(*
Nazwa:			FB_WickFeederStation
Opis:			Podajnik knotów
Wersja:			v1.0
Data:			2025-12-29
Autor:			MK
Urzadzenia:		Podnosnik stacji, grzałka, czujnik temp, ssawka
Konfiguracja:	
Info: 
*)




FUNCTION_BLOCK FB_WickFeederStation
VAR_INPUT
	_CONTROL_:BOOL;	
	bEnable:BOOL;					//Zezowlenie na pracę podajnika knotów
	bEStop:BOOL;					//Stop awaryjny nieaktywny
	bRun:BOOL;						//Zezwolenie na podanie knotów do wbijaków - jak maszyna w Execute musi być na 1
	bRun1: BOOL;					//Zezwolenie na wbicie knota
	bRun2: BOOL;					//Zezwolenie na wbicie knota
	bHoming:BOOL;					//Zezwolenie na wykonanie bazowania i pozycjonowania podajnika
	bHeightSet:BOOL;				//Ustaw wysokość
	bIgnoreError:BOOL;				//Ignorowania błędów cyklu pracy
	bReset:BOOL;					//Reset błędu, jeśli w stanie "eError"
	lrPositionHeightSV:LREAL;		//Wysokość zadana na której ma znajdować się podajnik
	lrMaxHeight:LREAL;				//Maksymalna wysokość podajnika platynek
	lrMinHeight:LREAL;				//Minimalna wysokość podajnika platynek
	bManualMovement:BOOL; 			//Uruchomienie trybu ruchów ręcznych
	
	_SENSORS_:BOOL;	
	bWheelLevelSensor			: BOOL;	
	bWheelSensor				: BOOL;
	bQueFullAfterWheelSensor	: BOOL;			//Czujnik zapełnienia rękawa
	bQueFullSensor				: BOOL;			//Czujnik zapełnienia rękawa
	bWickAtPipe					: BOOL;			//Czujnik na końcu rękawa
	bSeparatorPos1				: BOOL;			//Separator nad torem 1
	bSeparatorPos2				: BOOL;			//Separator nad torem 2
	bQueFullAtSleve1			: BOOL;			//Czujnik zapełnienia rękawa 1
	bQueFullAtSleve2			: BOOL;			//Czujnik zapełnienia rękawa 2
	bWickAtSleve1				: BOOL;			//Czujnik na końcu rękawa 1
	bWickAtSleve2				: BOOL;			//Czujnik na końcu rękawa 2
	bSleve1SeparatorIn			: BOOL;			//Separator pod rękawem
	bSleve1SeparatorOut			: BOOL;			//Separator nad butelką
	bSleve2SeparatorIn			: BOOL;			//Separator pod rękawem
	bSleve2SeparatorOut			: BOOL;			//Separator nad butelką
	bHammer1Up					: BOOL;			//Wbijak pozycja górna
	bHammer1Down				: BOOL;			//Wbijak pozycja dolna
	bHammer2Up					: BOOL;			//Wbijak pozycja górna
	bHammer2Down				: BOOL;			//Wbijak pozycja dolna
	bFormPositioningHide1		: BOOL;			//Wbijak pozycja dolna
	bFormPositioningHide2		: BOOL;			//Wbijak pozycja dolna
	
	_HEIGHTMOTOR_ :BOOL;	
	udiHeightMotorEncoderCV		: UDINT;		//Sygnał impulsów enkodera siłownika
	bHeightEncoderSetCDone		: BOOL;	
	rHeightMotorPositionOffset 	: REAL;			//Wysokość bazowani podnośnika
//	nPositionHeightCV			: LREAL;		//Aktualna wysokość podajnika platynek
	
	_BOWLMOTOR_ :BOOL;
	bEngineOK					: BOOL;					//Wejście czujnika zabezpieczenia silnika 
	InEngineVelocityCV 			: UDINT;		
	InEngineSTW 				: UINT; 				// Statusword transportera wejściowo wyjściowego
	IbEngineWcState				: BOOL; 				// Statusword transportera wejściowo wyjściowego
	_PARAMETERS_:BOOL;
	iTimeDelayOn				: INT; 					//Czas na właczenie silnika sortera po zaniku sygnału przepełnienia z rękawa
	iTimeDelayOff				: INT; 					// Czas na wylączenie silnika sortera po wykryciu sygnału przepełnienia z rękawa sortera
	iTimeToEmptySleeveError		: INT;					// Czas do włączenia alrmu pustego rękawa

	_ALARMINFO_ :BOOL;
	iStationIndex:UDINT;					//Numer stacji 
	sStationName:WSTRING;					//Nazwa stacji	

	
END_VAR
VAR_OUTPUT
	eState: E_Station;						//Stan ogólny bloku
	eRunningStateFeeder: E_WickFeederSorterState;		//Stan podajnika platynek
	eRunningState1: E_WickFeederState;		//Stan podajnika platynek
	eRunningState2: E_WickFeederState;		//Stan podajnika platynek
	
	bError: BOOL;							//Błąd stacji
	nErrorNr: UDINT;						//Nr błędu podajnika platynek
	sErrorDescription:STRING(200);			//Opis błędu
	sErrorDescription2: STRING(200);		//Opis błędu 2
	sErrorStationName:STRING;				//Nazwa stacji
	udiStationID:UDINT;						// Nr stacji
	
	tCycleTime:TIME;	
	bHomingDone:BOOL;						//Wymagane ponowne bazowanie (blad podczas bazowania lub stop awaryjny)	
	bCycleDone1	:BOOL;
	bCycleDone2	:BOOL;
	bCycleNotDone1:BOOL;
	bCycleNotDone2:BOOL;
	
	bHeightMotorUp				:BOOL;					//Sterowanie silnikiem podnośnika  - RUCH W GÓRĘ
	bHeightMotorDown			:BOOL;					//Sterowanie silnikiem podnośnika  - RUCH W DÓŁ
	lrHeightMotorCV				:LREAL;					//Aktualna pozycja podnośnika
	udiHeightMotorEncoderSetCV	: UDINT;		
	bHeightEncoderSetC			: BOOL;					// Zerowanie enkodera
	
	bSorterEngine 				: BOOL; 				// Sterowanie silnikiem sortera
	QnEngineVelocitySV 			: UDINT; 				// Nastawa prędkości
	QnEngineCTW 				: UINT;  				// Controlword transportera we/wy	
	
	bStopper1					: BOOL;			//Stoper1 przed separatorem
	bStopper2					: BOOL;			//Stoper2 przed separatorem
	bSeparator1					: BOOL;			//Separator nad torem 1
	bSeparator2					: BOOL;			//Separator nad torem 2
	bSleve1SeparatorActIn		: BOOL;			//Separator pod rękawem
	bSleve1SeparatorActOut		: BOOL;			//Separator nad butelką
	bSleve2SeparatorActIn		: BOOL;			//Separator pod rękawem
	bSleve2SeparatorActOut		: BOOL;			//Separator nad butelką
	bHammer1					: BOOL;			//Wbijak 
	bHammer2					: BOOL;			//Wbijak
	bFormPositioning			: BOOL;			//Pozycjonowanie 1
	bBlow1						: BOOL;
	bSleeveBlow					: BOOL;
	
	bWarning					: BOOL;
END_VAR

VAR_IN_OUT
	bManualHeightMotorUp		: BOOL;					//Ruch ręczny podnośnika stacji w górę
	bManualHeightMotorDown		: BOOL;					//Ruch ręczny podnośnika stacji w dół
	bManualSorterEngine			: BOOL;					//Ręczne włączenie silnika sortera
	bManualSorterAir			: BOOL;					//Ręczne włączenie zaworu wydmuchu
	
	bManualStopper				: BOOL;		
	bManualStopper2				: BOOL;						
	bManualSeparator1			: BOOL;			//Separator nad torem 1
	bManualSeparator2			: BOOL;			//Separator nad torem 2
	bManualSleve1SeparatorActIn	: BOOL;			//Separator pod rękawem
	bManualSleve1SeparatorActOut: BOOL;			//Separator nad butelką
	bManualSleve2SeparatorActIn	: BOOL;			//Separator pod rękawem
	bManualSleve2SeparatorActOut: BOOL;			//Separator nad butelką
	bManualHammer1				: BOOL;			//Wbijak 
	bManualHammer2				: BOOL;			//Wbijak					
	bManualFormPositioning		: BOOL;			//Wbijak	
END_VAR

VAR
	//Podnośnik Jiesang	
	fbHeightMotorEncoder: FB_JiesangActuatorEncoderModul;	// Blok enkodera podnośnika chwytaka stabilizującego pod zakręcarką	
	bHeightMotorEncoderCounterReset:BOOL; 				//Sygnał resetu enkodera
	bHeightMotorEncoderHomed:BOOL;						//Informacja od enkodera że jest zbazowany
	lrLastPositionHeightCV			: LREAL;			//Pozycja podnośnika w poprzednim cyklu programu
	
	
	fbInverter: FB_MitsubishiInverter;
	tonInverterError: TON;

	
	eLastState: E_Station;							//Stan ogólny bloku
	eLastRunningState: E_WickFeederState;			//Stan podbloku
	eLastStateTemp: E_Station;						//Stan ogólny bloku
	eLastRunningStateTemp: E_WickFeederState;		//Stan podbloku
	bStateError: BOOL;
	tonEstopDelay: TON;
	
	
	
	bManualPositionChanged						: BOOL;
	
	tonHomingSensor								: TON;
	tonHeightNoChange			: TON; 					// Timer wykrycia braku ruchu siłownika zmiany wysokości stacji
	tonHeightNoChangeTime		: TON; 					// Timer wykrycia braku ruchu siłownika zmiany wysokości stacji
	tofHeightMotorDown			: TOF;
	tofHeightMotorUp			: TOF;
	
	tonLimitPosMinReachedDelay	: TON;					// Timer osoiągniecia minimalnej wyskości 
	tonLimitPosMaxReachedDelay	: TON;					// Timer osiągnięcia maksymalnej wyskości
	tonSortingEngineOn			: TON;					// Opóźnienie po załączeniu napędu
	tonSortingEngineOff			: TON;					// Opóźnienie wyłączenia napędu
	tonSleeveFullEngineOn		: TON;					// Czas załączenia napędu po wykrciu braku nasadek
	tonEngineBlocked			: TON;					// Zablokowany silnik	
	tonTryUnblockWheel			: TON;					// Czas ruchu falownika w drugą stronę
	
	tonAirBeforeStart			: TON;					// Czasówka opóźeniani przedmuchu
	tonAirBeforeStart2			: TON;					// Czasówka opóźeniani przedmuchu
	tonAirAfterStop				: TON;					// Czasówka przedmuchu po zatrzymaniu
	tonStoppingTime				: TON;					// Czasówka zbyt długiego zatrzymawania
	
	rtEncoderHomed				: R_TRIG;				// Bit zakończenia enkodera
	rtWheelSensor				: R_TRIG;
	bTryUnblockWheel 			: BOOL;
	iTryUnblockWheel 			: INT;
	
	TimerOn						: TON;
	TimerOff					: TON;
	bImpOn						: BOOL;
	
	tonHammer1Down				: TON;
	tonHammer2Down				: TON;
	
	tonErrorHeightChange		: TON; 					// Timer błędu zacięcia się podnośnika
	tonEmptySleeveError			: TON;					// Timer pustego rękawa
	tonMaxHeightError			: TON;					// Timer ustawienia zbyt dużej wysokości stacji
	tonMinHeightError			: TON;					// Timer ustawienia zbyt małej wysokości stacji
	tonSorterEngineError		: TON;
	tonbSeparatorPos1AndNotbWickAtSleve1 : TON;	
	tonbSeparatorPos2AndNotbWickAtSleve2 : TON;		
	tonbSeparatorPos1 : TON;
	tonbSeparatorPos2 : TON;
	tonbWickAtPipe : TON;
	tobbSleve1SeparatorIn : TON;
	tobbSleve2SeparatorIn : TON;

	tonSeparatorPos1Error		: TON;
	tonSeparatorPos2Error		: TON;
	tonSleve1SeparatorInError	: TON;
	tonSleve1SeparatorOutError	: TON;
	tonSleve2SeparatorInError	: TON;
	tonSleve2SeparatorOutError	: TON;
	tonHammer1UpError			: TON;
	tonHammer1DownError			: TON;
	tonHammer2UpError			: TON;
	tonHammer2DownError			: TON;
	tonWickBlocked1				: TON;
	tonWickBlocked2				: TON;
	
	
	//Zmienne od EVENTLOGGER
	bAlarmInit 						: BOOL := TRUE; 
	nAlarmNumerator					: INT;
	arfbAlarm						: ARRAY[0..19] OF  FB_TcAlarm;		//Tablica bloczków błędów
	fbSourceInfo 					: FB_TcSourceInfo;
	iSourceInfo						: I_TcSourceInfo;
	sAlarmTest						: STRING;
	//Koniec zmiennych od EVENTLOGGER

	rtbSeparator1: R_TRIG;
	rtbSeparator2: R_TRIG;
	rtbSleve1SeparatorActIn: R_TRIG;
	rtbSleve1SeparatorActOut: R_TRIG;
	rtbSleve2SeparatorActIn: R_TRIG;
	rtbSleve2SeparatorActOut: R_TRIG;
	fbbQueFullAtSleve1: FB_InputFilter_v2;
	fbbQueFullAtSleve2: FB_InputFilter_v2;	
	fbbWickAtPipe: FB_InputFilter_v2;
	fbbNotWickAtPipe: FB_InputFilter_v2;	
	iSortingCase: INT;
	tonCaseA: TON;
	tonCaseB: TON;	
	tonCaseC: TON;	
	tonCaseD: TON;
	bSeparatorLast:BOOL;
	bWickBlocked:BOOL;
	tonLowLevelSensor:TON;
END_VAR


ACT_HeightMotor();
ACT_ErrorHandling();
ACT_Warning();
ACT_Inverter();
ACT_Control();
ACT_Signals();
//Statistics();
//EncoderTest();
//aStationID();
(*Zapisywanie ostatniego stanu*)
// IF eLastStateTemp<>eState THEN
// 	eLastState := eLastStateTemp;
// END_IF
// eLastStateTemp := eState;
// IF eLastRunningStateTemp<>eRunningState THEN
// 	eLastRunningState := eLastRunningStateTemp;
// END_IF
// eLastRunningStateTemp := eRunningState;
(*Koniec Zapisywanie ostatniego stanu*)

lrLastPositionHeightCV:=lrHeightMotorCV;

ACTION ACT_Control:
	(*****Wyłączenie enable*****)
	IF NOT bEnable THEN
		IF eState <> E_Station.eDisabled AND eState <> E_Station.ePreparingToDisable THEN
				eState 				:= E_Station.ePreparingToDisable; 
		END_IF	
	END_IF

	(*****Estop*****)
	IF NOT bEstop  THEN	
		IF eState <> E_Station.eAborted AND eState <> E_Station.eAborting AND eState <> E_Station.eDisabled THEN
				eState 				:= E_Station.eAborting; 
		END_IF
	END_IF


	CASE eState OF
//--------------------------------------------------------------------------------
// Stan maszyny po wyłączeniu i przygotowanie do uruchomienia
	E_Station.eDisabled: 					// Stan nieaktywnosci (Stacja wyłączona) 
	
		IF bEnable THEN
			eState 				:= E_Station.ePreparingToReady; 
		END_IF 
		
//--------------------------------------------------------------------------------
// Stan maszyny po zatrzymaniu awaryjnym   
	E_Station.eAborted: 					// Stan bezpiecznego zatrzymania (po Abortingu) 

		IF bEStop THEN
			eState 				:= E_Station.ePreparingToReady;
		END_IF
		
//--------------------------------------------------------------------------------
// Stan maszyny naciśnieciu estopa 	
	E_Station.eAborting:                 	// Stan bezpiecznego zatrzymywania (po EStopie)
// 		bGate1:= FALSE;
// 		bGate2:= FALSE;
	
		ACT_ResetCommands();

		eState 						:=  E_Station.eAborted;  
		//eRunningState				:=	E_LidFeederState.eReady;
		
//--------------------------------------------------------------------------------
// Stan masyzny po wykryciu błędu			
	E_Station.eError:                 	 	// Stan błędu 	
		
		ACT_ResetCommands();
		
		IF bReset THEN
			eState 				:= E_Station.eResetting;
			bError := FALSE;
		END_IF
		
//--------------------------------------------------------------------------------
// Stan masyzny po wykryciu błędu
	E_Station.eResetting:					// Stan resetowania bledu (po Errorze)
// 			CASE udiErrorID-udiStationIndex OF
// 		
// 				//Error 8 - Błąd falownika
// 				9:
// 					fbInverter.bReset	:= TRUE;
// 					bError 				:= FALSE;
// 				ELSE
// 					bError := FALSE;	
// 			END_CASE		
		
		IF NOT bError AND fbInverter.eState = E_Station.eReady THEN
			fbInverter.bReset	:= FALSE;	
			{warning 'Sprawdzić błąd falownika CapFeeder'}
			nErrorNr 			:=	0;
			sErrorDescription 	:=	'';
			eState 				:=	E_Station.ePreparingToReady;
			//eRunningState		:=	E_CapFeederState.eReady;
		ELSE
			eState 				:=	E_Station.eError;
		END_IF
    
//--------------------------------------------------------------------------------
// Stan ruchoow manualnych
	E_Station.eManualMovement:     			// Stan ruchów manualnych  
   
		ACT_ManualMovements();
		IF bManualHeightMotorUp OR bManualHeightMotorDown OR bSeparator1 OR bSeparator2 OR 
			bSleve1SeparatorActIn OR bSleve2SeparatorActIn OR bSleve1SeparatorActOut OR bSleve2SeparatorActOut THEN
				//bManualPositionChanged		:= TRUE;
			END_IF
		//Wyjście z trybu serwisowego
		IF NOT bManualMovement THEN
			
			bHeightMotorUp				:=	FALSE;
			bHeightMotorDown			:=	FALSE;
			bStopper1					:= FALSE;
			bStopper2					:= TRUE;			
 			bSeparator1					:= FALSE;
 			bSeparator2					:= FALSE;
 			bSleve1SeparatorActIn		:= FALSE;  
 			bSleve1SeparatorActOut	    := FALSE;
 			bSleve2SeparatorActIn	    := FALSE;
 			bSleve2SeparatorActOut	    := FALSE;
 			bHammer1				    := FALSE;
 			bHammer2				    := FALSE;
			bBlow1						:= FALSE;
			bSleeveBlow						:= FALSE;
			bFormPositioning			:= FALSE;
			
			IF bManualPositionChanged THEN
				bHomingDone				:= FALSE;
				bManualPositionChanged	:= FALSE;
			END_IF
			
			eState:=E_Station.eReady;
		END_IF
		

//--------------------------------------------------------------------------------
// Stan rozpoczecia bazowania
	E_Station.eHoming:						// Stan bazowania 
		
		ACT_Homing();
		IF NOT bHoming AND NOT bHeightSet THEN
			bHeightMotorDown					:=	FALSE;
			bHeightMotorUp						:=	FALSE;
		   eState								:=E_Station.ePreparingToReady;
		END_IF		
		
//--------------------------------------------------------------------------------
// Stan zakończenia bazowania
	E_Station.eHomingDone:                  // Stan wykonania bazowania 
	
		bHeightMotorDown					:=	FALSE;
		bHeightMotorUp						:=	FALSE;
		//bHeightMotorEncoderCounterReset		:=	FALSE;
		bHomingDone							:=	TRUE;
		IF NOT bHoming AND NOT bHeightSet THEN
		   eState:=E_Station.eReady;
		END_IF
		
//--------------------------------------------------------------------------------
// Stan przygotowania do gotowości
	E_Station.ePreparingToReady:            // Stan przygotowywania do gotowosci (zawsze przed Ready)  
		

		bStopper2							:=	TRUE;		
		bSorterEngine						:=	FALSE;

		eState								:=	E_Station.eReady;	
		eRunningState1						:=	E_WickFeederState.eReady;
		eRunningState2						:=	E_WickFeederState.eReady;		
//-------------------------------------------------------------------------------
// Stan przygotowania do wyłączenia maszyny
	E_Station.ePreparingToDisable:          // Stan przygotowywania do nieaktywnosci (po wyłączeniu Enable) 
		
// 		bGate1:= FALSE;
// 		bGate2:= FALSE;
		bHomingDone									:= FALSE;	
		bSorterEngine:=FALSE;
//		bSorterAir:=FALSE;
		bHeightMotorUp:= NOT tonHomingSensor.Q;
		bHeightMotorDown:=FALSE;	
		IF tonHeightNoChange.Q OR tonHeightNoChangeTime.Q THEN
			bHeightMotorUp			:=	FALSE;
			bHeightMotorDown		:=	FALSE;	
			//eRunningState			:=	E_CapFeederState.eReady;		
			eState					:=	E_Station.eDisabled;
		END_IF	
			
//--------------------------------------------------------------------------------
// Stan gotowości
	E_Station.eReady:						// Stan gotowosci 
	
		IF bRun  THEN
			eState 				:= E_Station.eStarting; 
		END_IF
		IF bHoming OR bHeightSet THEN
			bHomingDone							:=	FALSE;
			eState 								:= E_Station.eHoming; 
		END_IF
		IF bManualMovement THEN
			//Jeśli przejście w tryb ruchów manualnych przepisz wszystkie stany siłowników sterowanych przez moduł
			//aby zapobiec ewentualnym kolizjom po wejściu w tryb serwisowy
			fbInverter.bDirection 		:= TRUE;
		
			bManualPositionChanged		:= FALSE;
			bHeightMotorUp				:= bManualHeightMotorUp;
			 bManualHeightMotorDown		:=	bHeightMotorDown		;
			 bManualSorterEngine        :=	bSorterEngine			;
			 bManualSorterAir           :=	bBlow1					;
			 bManualSorterAir            :=	bSleeveBlow					;
			 bManualStopper                 :=	bStopper1			;	
			 bManualStopper2	                    :=	bStopper2	;			
			 bManualSeparator1			        :=    bSeparator1	;			
			 bManualSeparator2                   :=    bSeparator2	;			
			 bManualSleve1SeparatorActIn         :=    bSleve1SeparatorActIn	;
    		 bManualSleve1SeparatorActOut        :=    bSleve1SeparatorActOut	;
    		 bManualSleve2SeparatorActIn         :=    bSleve2SeparatorActIn	;
    		 bManualSleve2SeparatorActOut        :=    bSleve2SeparatorActOut	;
    		 bManualHammer1                      :=    bHammer1				    ;
    		 bManualHammer2                      :=    bHammer2				    ;
			 bManualFormPositioning             :=	bFormPositioning		    ;
					
			eState 						:= E_Station.eManualMovement; 
		END_IF
		IF NOT bRun THEN
			bCycleDone1 		:= FALSE;
			bCycleNotDone1 		:= FALSE;	
			bCycleDone2 		:= FALSE;
			bCycleNotDone2 		:= FALSE;	
		END_IF
		IF NOT bRun1 THEN
			bCycleDone1 		:= FALSE;
			bCycleNotDone1 		:= FALSE;	
		END_IF	
		IF NOT bRun2 THEN
			bCycleDone2 		:= FALSE;
			bCycleNotDone2 		:= FALSE;	
		END_IF		
//--------------------------------------------------------------------------------
// Stan zatrzymywania
	E_Station.eStopping:					// Stan zatrzymywania 
		
//		bSorterAir 		:= 	TRUE;
		bSorterEngine 	:=	FALSE;
//		IF tonStoppingTime.Q AND eRunningState1=E_WickFeederSorterState.eReady AND eRunningState2=E_WickFeederSorterState.eReady THEN
		IF tonStoppingTime.Q  THEN
			
			ACT_ResetCommands();
			//eRunningState							:= E_CapFeederState.eReady;
			eState									:= E_Station.eReady;
		END_IF

		
//--------------------------------------------------------------------------------
// Stan uruchomienia lini ( po eReady)
	E_Station.eStarting:                  	// Stan uruchamiania (po Ready)
//		iValvesCycleCase		:=0;
		eState					 := E_Station.eRunning; 

//--------------------------------------------------------------------------------
// Stan wykonywania pracy
	E_Station.eRunning:               		// Stan wykonywania cyklu (po Startingu), w tym stanie osobny

		ACT_Running();
		IF NOT bRun THEN 					(*Przerywanie cyklu*)
			eState				:= E_Station.eStopping;
			//bCycleNotDone		:= TRUE;
		END_IF
		(*IF bCycleDone OR bCycleNotDone THEN (*Cykl zakończony*)
			eState 				 := E_Station.eReady;
		END_IF*)						
		
		
END_CASE
END_ACTION

ACTION ACT_ErrorHandling:
(*
Alarm_0620	620	Error	Blokada podnośnika lub brak zasilania - sprawdź czujnik lub odblokuj mechanicznie
Alarm_0621	621	Error	Pusty rękaw sortera - uzupełnij nasadki
Alarm_0622	622	Error	Wartość zadana wysokości jest większa od maksymalnej - zmień ustawienia w recepturze {0}
Alarm_0623	623	Error	Wartość zadana wysokości jest mniejsza od minimalnej - zmień ustawienia w recepturze {0}
Alarm_0624	624	Error	Błąd falownika
Alarm_0625	625	Error	Błąd siłownika rozdzielacza pozycja 1
Alarm_0626	626	Error	Błąd siłownika rozdzielacza pozycja 2
Alarm_0627	627	Error	Błąd wysunięcia siłownika separatora 1
Alarm_0628	628	Error	Błąd cofnięcia siłownika separatora 1
Alarm_0629	629	Error	Błąd wysunięcia siłownika separatora 2
Alarm_0630	630	Error	Błąd cofnięcia siłownika separatora 2
Alarm_0631	631	Error	Błąd wysunięcia wbijaka 1
Alarm_0632	632	Error	Błąd cofnięcia wbijaka 1
Alarm_0633	633	Error	Błąd wysunięcia wbijaka 2
Alarm_0634	634	Error	Błąd cofnięcia wbijaka 2
Alarm_0635	635	Error	Blokada knota w rękawie 1
Alarm_0636	636	Error	Blokada knota w rękawie 2
*)

IF bAlarmInit THEN
    bAlarmInit := FALSE; 
	fbSourceInfo.Clear();
	fbSourceInfo.sName:=wsLiteral_TO_UTF8(sStationName);//'Machine';
	fbSourceInfo.nId:=udiStationID;//2700;
	// Alarm_0620	620	Error	Blokada podnośnika lub brak zasilania - sprawdź czujnik lub odblokuj mechanicznie
    arfbAlarm[0].CreateEx(stEventEntry := TC_EVENTS.AlarmClass.Alarm_0620, bWithConfirmation:= FALSE,  ipSourceInfo:= fbSourceInfo); 
	// Alarm_0621	621	Error	Pusty rękaw sortera - uzupełnij nasadki
	arfbAlarm[1].CreateEx(stEventEntry := TC_EVENTS.AlarmClass.Alarm_0621, bWithConfirmation:= FALSE,  ipSourceInfo:= fbSourceInfo); 
	// Alarm_0622	622	Error	Wartość zadana wysokości jest większa od maksymalnej - zmień ustawienia w recepturze {0}
	arfbAlarm[2].CreateEx(stEventEntry := TC_EVENTS.AlarmClass.Alarm_0622, bWithConfirmation:= FALSE,  ipSourceInfo:= fbSourceInfo); 
	// Alarm_0623	623	Error	Wartość zadana wysokości jest mniejsza od minimalnej - zmień ustawienia w recepturze {0}
	arfbAlarm[3].CreateEx(stEventEntry := TC_EVENTS.AlarmClass.Alarm_0623, bWithConfirmation:= FALSE,  ipSourceInfo:= fbSourceInfo); 
	// Alarm_0624	624	Error	Błąd falownika
	arfbAlarm[4].CreateEx(stEventEntry := TC_EVENTS.AlarmClass.Alarm_0624, bWithConfirmation:= FALSE,  ipSourceInfo:= fbSourceInfo); 
	// Alarm_0625	625	Error	Błąd siłownika rozdzielacza pozycja 1
	arfbAlarm[5].CreateEx(stEventEntry := TC_EVENTS.AlarmClass.Alarm_0625, bWithConfirmation:= FALSE,  ipSourceInfo:= fbSourceInfo); 
	// Alarm_0626	626	Error	Błąd siłownika rozdzielacza pozycja 2
	arfbAlarm[6].CreateEx(stEventEntry := TC_EVENTS.AlarmClass.Alarm_0626, bWithConfirmation:= FALSE,  ipSourceInfo:= fbSourceInfo); 
	// Alarm_0627	627	Error	Błąd wysunięcia siłownika separatora 1
	arfbAlarm[7].CreateEx(stEventEntry := TC_EVENTS.AlarmClass.Alarm_0627, bWithConfirmation:= FALSE,  ipSourceInfo:= fbSourceInfo); 
	// Alarm_0628	628	Error	Błąd cofnięcia siłownika separatora 1
	arfbAlarm[8].CreateEx(stEventEntry := TC_EVENTS.AlarmClass.Alarm_0628, bWithConfirmation:= FALSE,  ipSourceInfo:= fbSourceInfo); 
	// Alarm_0629	629	Error	Błąd wysunięcia siłownika separatora 2
	arfbAlarm[9].CreateEx(stEventEntry := TC_EVENTS.AlarmClass.Alarm_0629, bWithConfirmation:= FALSE,  ipSourceInfo:= fbSourceInfo); 
	// Alarm_0630	630	Error	Błąd cofnięcia siłownika separatora 2
	arfbAlarm[10].CreateEx(stEventEntry := TC_EVENTS.AlarmClass.Alarm_0630, bWithConfirmation:= FALSE,  ipSourceInfo:= fbSourceInfo); 
	// Alarm_0631	631	Error	Błąd wysunięcia wbijaka 1
	arfbAlarm[11].CreateEx(stEventEntry := TC_EVENTS.AlarmClass.Alarm_0631, bWithConfirmation:= FALSE,  ipSourceInfo:= fbSourceInfo);
	// Alarm_0632	632	Error	Błąd cofnięcia wbijaka 1
	arfbAlarm[12].CreateEx(stEventEntry := TC_EVENTS.AlarmClass.Alarm_0632, bWithConfirmation:= FALSE,  ipSourceInfo:= fbSourceInfo);
	// Alarm_0633	633	Error	Błąd wysunięcia wbijaka 2
	arfbAlarm[13].CreateEx(stEventEntry := TC_EVENTS.AlarmClass.Alarm_0633, bWithConfirmation:= FALSE,  ipSourceInfo:= fbSourceInfo);
	// Alarm_0634	634	Error	Błąd cofnięcia wbijaka 2
	arfbAlarm[14].CreateEx(stEventEntry := TC_EVENTS.AlarmClass.Alarm_0634, bWithConfirmation:= FALSE,  ipSourceInfo:= fbSourceInfo);
	// Alarm_0635	635	Error	Blokada knota w rękawie 1
	arfbAlarm[15].CreateEx(stEventEntry := TC_EVENTS.AlarmClass.Alarm_0635, bWithConfirmation:= FALSE,  ipSourceInfo:= fbSourceInfo);
	// Alarm_0636	636	Error	Blokada knota w rękawie 2
	arfbAlarm[16].CreateEx(stEventEntry := TC_EVENTS.AlarmClass.Alarm_0636, bWithConfirmation:= FALSE,  ipSourceInfo:= fbSourceInfo);
END_IF


//OBSŁUGA BŁĘDÓW 
//tonEstopDelay			(IN:=bEstop,	PT:=T#5S); //Opóżnienie po EStopie w celu blokoady błędów, powietrze jest później niż Estop a sygnał z czujnika nie pokazuje braku powietrza bo jest odcinany za tym

//************LISTA BŁĘDÓW***************
bStateError:= (eState=E_Station.eError) OR (eState=E_Station.eResetting);(* OR bIgnoreError; *)
//Error 1 - podnośnik nie porusza się pomimo wysterowania 
tonErrorHeightChange(IN:=(bHeightMotorUp OR bHeightMotorDown) AND lrLastPositionHeightCV=lrHeightMotorCV, PT:=T#3S);
tonEmptySleeveError(IN:=NOT bQueFullSensor AND bRun, PT:=INT_TO_TIME(iTimeToEmptySleeveError)*1000); //Było 30, teraz jest z receptur
tonMaxHeightError(IN:=lrPositionHeightSV>lrMaxHeight AND NOT bHomingDone AND eState=E_Station.eReady,PT:=T#30S);
tonMinHeightError(IN:=lrPositionHeightSV<lrMinHeight AND NOT bHomingDone AND eState=E_Station.eReady,PT:=T#30S);
tonSorterEngineError(IN:= NOT bEngineOK AND bSorterEngine, PT:=T#3S);
tonInverterError(IN:=fbInverter.bError AND NOT bStateError, PT:=T#3S);

IF bEnable THEN
	// Alarm_0620	620	Error	Blokada podnośnika lub brak zasilania - sprawdź czujnik lub odblokuj mechanicznie
	IF tonErrorHeightChange.Q THEN
		IF NOT arfbAlarm[0].bActive THEN
			bHeightMotorUp:=FALSE;
			bHeightMotorDown:=FALSE;
			arfbAlarm[0].Raise(nTimeStamp:=0);
		END_IF
	ELSE	
		IF  arfbAlarm[0].bActive AND bReset THEN
			arfbAlarm[0].Clear(nTimeStamp:=0, bResetConfirmation:= FALSE);
		END_IF
	END_IF
	
	// Alarm_0621	621	Error	Pusty rękaw sortera - uzupełnij nasadki
	IF tonEmptySleeveError.Q THEN
		IF NOT arfbAlarm[1].bActive THEN
			arfbAlarm[1].Raise(nTimeStamp:=0);
		END_IF
	ELSE	
		IF  arfbAlarm[1].bActive AND bReset THEN
			arfbAlarm[1].Clear(nTimeStamp:=0, bResetConfirmation:= FALSE);
		END_IF
	END_IF
	
	// Alarm_0622	622	Error	Wartość zadana wysokości jest większa od maksymalnej - zmień ustawienia w recepturze {0}
	IF tonMaxHeightError.Q THEN
		arfbAlarm[2].ipArguments.Clear() .AddLReal(lrMaxHeight);
		IF NOT arfbAlarm[2].bActive THEN
// 			bHeightMotorUp:=FALSE;
// 			bHeightMotorDown:=FALSE;
			arfbAlarm[2].Raise(nTimeStamp:=0);
		END_IF
	ELSE	
		IF  arfbAlarm[2].bActive AND bReset THEN
			arfbAlarm[2].Clear(nTimeStamp:=0, bResetConfirmation:= FALSE);
		END_IF
	END_IF
	
	// Alarm_0623	623	Error	Wartość zadana wysokości jest mniejsza od minimalnej - zmień ustawienia w recepturze {0}
		IF tonMinHeightError.Q THEN
			arfbAlarm[3].ipArguments.Clear() .AddLReal(lrMinHeight);
		IF NOT arfbAlarm[3].bActive THEN
// 			bHeightMotorUp:=FALSE;
// 			bHeightMotorDown:=FALSE;
			arfbAlarm[3].Raise(nTimeStamp:=0);
		END_IF
	ELSE	
		IF  arfbAlarm[3].bActive AND bReset THEN
			arfbAlarm[3].Clear(nTimeStamp:=0, bResetConfirmation:= FALSE);
		END_IF
	END_IF
	
	// Alarm_0624	624	Error	Błąd falownika
	IF tonInverterError.Q THEN
		IF NOT arfbAlarm[4].bActive THEN
			arfbAlarm[4].Raise(nTimeStamp:=0);
		END_IF
		IF arfbAlarm[4].bActive AND bReset THEN
			fbInverter.bReset := TRUE;
		END_IF
	ELSE	
		IF  arfbAlarm[4].bActive AND bReset THEN
			arfbAlarm[4].Clear(nTimeStamp:=0, bResetConfirmation:= FALSE);
		END_IF
	END_IF			

	// Alarm_0625	625	Error	Błąd siłownika rozdzielacza pozycja 1
	tonSeparatorPos1Error(IN:=(bSeparator1 AND NOT bSeparatorPos1 ),PT:= T#2S(*T#2S*)); 
	IF tonSeparatorPos1Error.Q THEN
		IF NOT arfbAlarm[5].bActive THEN
			bSeparator1:=FALSE;	
			arfbAlarm[5].Raise(nTimeStamp:=0);
		END_IF
	ELSE	
		IF  arfbAlarm[5].bActive AND bReset THEN
			arfbAlarm[5].Clear(nTimeStamp:=0, bResetConfirmation:= FALSE);
		END_IF
	END_IF;
	// Alarm_0626	626	Error	Błąd siłownika rozdzielacza pozycja 2
	tonSeparatorPos2Error(IN:=(bSeparator2 AND NOT bSeparatorPos2 ),PT:= T#2S); 
	IF tonSeparatorPos1Error.Q THEN
		IF NOT arfbAlarm[6].bActive THEN
			bSeparator2:=FALSE;	
			arfbAlarm[6].Raise(nTimeStamp:=0);
		END_IF
	ELSE	
		IF  arfbAlarm[6].bActive AND bReset THEN
			arfbAlarm[6].Clear(nTimeStamp:=0, bResetConfirmation:= FALSE);
		END_IF
	END_IF;	
	// Alarm_0627	627	Error	Błąd wysunięcia siłownika separatora 1
	tonSleve1SeparatorInError(IN:=bSleve1SeparatorActIn AND NOT bSleve1SeparatorIn,PT:= T#2S);	
	IF tonSleve1SeparatorInError.Q THEN
		IF NOT arfbAlarm[7].bActive THEN
			bSleve1SeparatorIn:=FALSE;	
			arfbAlarm[7].Raise(nTimeStamp:=0);
		END_IF
	ELSE	
		IF  arfbAlarm[7].bActive AND bReset THEN
			arfbAlarm[7].Clear(nTimeStamp:=0, bResetConfirmation:= FALSE);
		END_IF
	END_IF;	
	// Alarm_0628	628	Error	Błąd cofnięcia siłownika separatora 1
	tonSleve1SeparatorOutError(IN:=bSleve1SeparatorActOut AND NOT bSleve1SeparatorOut,PT:= T#2S);
	IF tonSleve1SeparatorOutError.Q THEN
		IF NOT arfbAlarm[8].bActive THEN
			bSleve1SeparatorOut:=FALSE;	
			arfbAlarm[8].Raise(nTimeStamp:=0);
		END_IF
	ELSE	
		IF  arfbAlarm[8].bActive AND bReset THEN
			arfbAlarm[8].Clear(nTimeStamp:=0, bResetConfirmation:= FALSE);
		END_IF
	END_IF;
	// Alarm_0629	629	Error	Błąd wysunięcia siłownika separatora 2
	tonSleve2SeparatorInError(IN:=bSleve2SeparatorActIn AND NOT bSleve2SeparatorIn,PT:= T#2S);	
	IF tonSleve2SeparatorInError.Q THEN
		IF NOT arfbAlarm[9].bActive THEN
			bSleve2SeparatorIn:=FALSE;	
			arfbAlarm[9].Raise(nTimeStamp:=0);
		END_IF
	ELSE	
		IF  arfbAlarm[9].bActive AND bReset THEN
			arfbAlarm[9].Clear(nTimeStamp:=0, bResetConfirmation:= FALSE);
		END_IF
	END_IF;	
	// Alarm_0630	630	Error	Błąd cofnięcia siłownika separatora 2
	tonSleve2SeparatorOutError(IN:=bSleve2SeparatorActOut AND NOT bSleve2SeparatorOut,PT:= T#2S);
	IF tonSleve2SeparatorOutError.Q THEN
		IF NOT arfbAlarm[10].bActive THEN
			bSleve2SeparatorOut:=FALSE;	
			arfbAlarm[10].Raise(nTimeStamp:=0);
		END_IF
	ELSE	
		IF  arfbAlarm[10].bActive AND bReset THEN
			arfbAlarm[10].Clear(nTimeStamp:=0, bResetConfirmation:= FALSE);
		END_IF
	END_IF;
	// Alarm_0631	631	Error	Błąd wysunięcia wbijaka 1
	tonHammer1DownError(IN:= bHammer1 AND NOT bHammer1Down ,PT:= T#2S);
	IF tonHammer1DownError.Q THEN
		IF NOT arfbAlarm[11].bActive THEN
			bHammer1:=FALSE;	
			arfbAlarm[11].Raise(nTimeStamp:=0);
		END_IF
	ELSE	
		IF  arfbAlarm[11].bActive AND bReset THEN
			arfbAlarm[11].Clear(nTimeStamp:=0, bResetConfirmation:= FALSE);
		END_IF
	END_IF;
	// Alarm_0632	632	Error	Błąd cofnięcia wbijaka 1
	tonHammer1UpError(IN:= NOT bHammer1 AND NOT bHammer1Up,PT:= T#2S);
	IF tonHammer1UpError.Q THEN
		IF NOT arfbAlarm[12].bActive THEN
			bHammer1:= TRUE;	
			arfbAlarm[12].Raise(nTimeStamp:=0);
		END_IF
	ELSE	
		IF  arfbAlarm[12].bActive AND bReset THEN
			arfbAlarm[12].Clear(nTimeStamp:=0, bResetConfirmation:= FALSE);
		END_IF
	END_IF;
	// Alarm_0633	633	Error	Błąd wysunięcia wbijaka 2
	tonHammer2DownError(IN:= bHammer2 AND NOT bHammer2Down ,PT:= T#2S);
	IF tonHammer2DownError.Q THEN
		IF NOT arfbAlarm[13].bActive THEN
			bHammer2:=FALSE;	
			arfbAlarm[13].Raise(nTimeStamp:=0);
		END_IF
	ELSE	
		IF  arfbAlarm[13].bActive AND bReset THEN
			arfbAlarm[13].Clear(nTimeStamp:=0, bResetConfirmation:= FALSE);
		END_IF
	END_IF;
	// Alarm_0634	634	Error	Błąd cofnięcia wbijaka 2
	tonHammer2UpError(IN:= NOT bHammer2 AND NOT bHammer2Up,PT:= T#2S);
	IF tonHammer2UpError.Q THEN
		IF NOT arfbAlarm[14].bActive THEN
			bHammer2:=TRUE;	
			arfbAlarm[14].Raise(nTimeStamp:=0);
		END_IF
	ELSE	
		IF  arfbAlarm[14].bActive AND bReset THEN
			arfbAlarm[14].Clear(nTimeStamp:=0, bResetConfirmation:= FALSE);
		END_IF
	END_IF;
	// Alarm_0635	635	Error	Blokada knota w rękawie 1
	tonWickBlocked1(IN:=bQueFullAfterWheelSensor AND NOT bQueFullSensor AND bRun, PT:=T#15S);
	IF tonWickBlocked1.Q THEN
		IF NOT arfbAlarm[15].bActive THEN
	
			arfbAlarm[15].Raise(nTimeStamp:=0);
		END_IF
	ELSE	
		IF  arfbAlarm[15].bActive AND bReset THEN
			arfbAlarm[15].Clear(nTimeStamp:=0, bResetConfirmation:= FALSE);
		END_IF
	END_IF;
	// Alarm_0636	636	Error	Blokada knota w rękawie 2
	tonWickBlocked2();
		IF tonWickBlocked2.Q THEN
		IF NOT arfbAlarm[16].bActive THEN
	
			arfbAlarm[16].Raise(nTimeStamp:=0);
		END_IF
	ELSE	
		IF  arfbAlarm[16].bActive AND bReset THEN
			arfbAlarm[16].Clear(nTimeStamp:=0, bResetConfirmation:= FALSE);
		END_IF
	END_IF;


ELSE
		bError 					:= FALSE;
END_IF
//*******KONIEC LISTA BŁĘDÓW***************


//******************PRZEJŚCIE DO eERROR*****************************

IF bError AND NOT bStateError THEN
// 	IF eLastState = eRunning THEN
// 		bCycleNotDone := TRUE;
// 	END_IF
	eState := E_Station.eError;
END_IF

//****************WYŚWIETLANIE STATUSU BLEDU***********************


(*Wyświetlanie błedu na wyjściu*)
bError							:= FALSE;
FOR nAlarmNumerator := 0 TO 19 DO
	bError						:= bError OR arfbAlarm[nAlarmNumerator].bActive;
END_FOR

(*Przepisywanie nazwy stacji*)
//sErrorStationName:=sStationName;



//Jezeli nie zbazowane to potrzebne bazowanie
IF NOT bHeightMotorEncoderHomed  THEN
	bHomingDone:=FALSE;
END_IF
END_ACTION

ACTION ACT_HeightMotor:
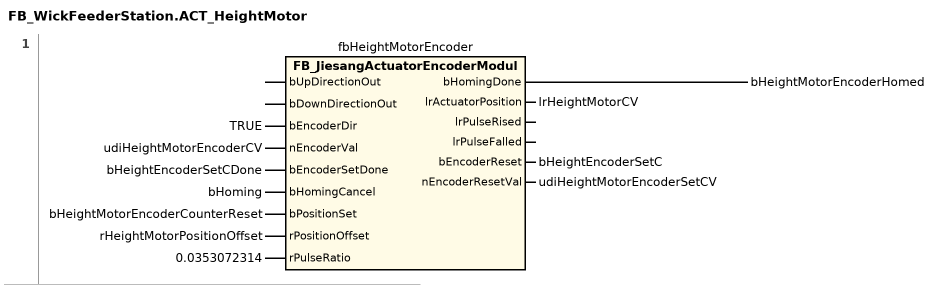
// NETWORK 1
fbHeightMotorEncoder(
    bEncoderDir := TRUE,
    nEncoderVal := udiHeightMotorEncoderCV,
    bEncoderSetDone := bHeightEncoderSetCDone,
    bHomingCancel := bHoming,
    bPositionSet := bHeightMotorEncoderCounterReset,
    rPositionOffset := rHeightMotorPositionOffset,
    rPulseRatio := 0.0353072314,
    lrActuatorPosition => lrHeightMotorCV,
    bEncoderReset => bHeightEncoderSetC,
    nEncoderResetVal => udiHeightMotorEncoderSetCV); // FB_JiesangActuatorEncoderModul
bHeightMotorEncoderHomed := fbHeightMotorEncoder.bHomingDone;
END_ACTION

ACTION ACT_Homing:
//BAZOWANIE

tofHeightMotorDown	(IN:=bHeightMotorDown, PT:=T#1S);	//Zabezpieczenie przed zbyt szybkim przełączeniem pomiędzy Down a Up, bezpiecznieki sie palą
tofHeightMotorUp	(IN:=bHeightMotorUp, PT:=T#1S); 	//Zabezpieczenie przed zbyt szybkim przełączeniem pomiędzy Down a Up, bezpiecznieki sie palą
//Ustaw siłowniki
bStopper1					:= TRUE; //Raczej zablokuj ?
bStopper2					:= TRUE;
//Do zastanowienia
bSeparator1					;
bSeparator2					;
//Podnieś wbijacze
bHammer1					:= FALSE;
bHammer2					:= FALSE;
//Wyłącz odmuchy
bBlow1						:= FALSE;
bSleeveBlow					:= FALSE;
bFormPositioning			:= FALSE;
//Jak wbijacze w górze to ustaw separator na załadunek
IF bHammer1Up THEN
	bSleve1SeparatorActIn	:= TRUE;
	bSleve1SeparatorActOut	:= FALSE;
END_IF

IF bHammer2Up THEN
	bSleve2SeparatorActIn	:= TRUE;
	bSleve2SeparatorActOut	:= FALSE;
END_IF

	
//Podnoszenie stacji do maksymalnej pozycji
IF NOT bHeightMotorEncoderHomed OR rtEncoderHomed.Q THEN
	bHeightMotorUp:= NOT tofHeightMotorDown.Q AND NOT tonHomingSensor.Q;
	bHeightMotorDown:= FALSE;
	IF tonHeightNoChange.Q THEN//OR tonHeightNoChangeTime.Q THEN
		bHeightMotorEncoderCounterReset:=TRUE;
		bHeightMotorUp:=FALSE;
   END_IF
	//Jesli enkoder zbazowany zakończ bazowanie	
	IF rtEncoderHomed.Q  THEN
		bHeightMotorUp:=FALSE;
		bHeightMotorDown:=FALSE;
		eState:=E_Station.eHomingDone;
	END_IF		
		
//Po podniesieniu stacji opuszczanie do ustalonej wysokości
ELSIF bHeightMotorEncoderHomed THEN
	bHeightMotorEncoderCounterReset:=FALSE;
	bHeightMotorUp:=lrHeightMotorCV<=lrPositionHeightSV;
	bHeightMotorDown:=lrHeightMotorCV>=lrPositionHeightSV;
	//Kiedy stacja osiągnie wysokość zadaną
	IF ABS(lrHeightMotorCV-lrPositionHeightSV)<0.5 OR tonLimitPosMaxReachedDelay.Q OR tonLimitPosMinReachedDelay.Q THEN
		bHeightMotorDown:=FALSE;
		bHeightMotorUp:=FALSE;
		//Jak siłowniki na miejscach
		IF bHammer1Up AND bHammer2Up AND bSleve1SeparatorIn AND bSleve2SeparatorIn THEN
			eState:=E_Station.eHomingDone;
		END_IF
	END_IF			
END_IF
END_ACTION

ACTION ACT_Inverter:
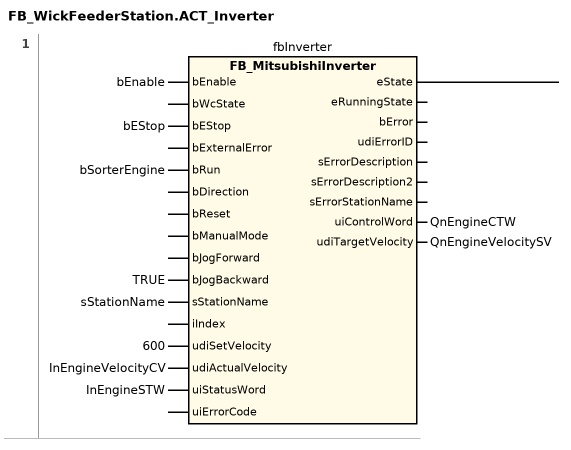
// NETWORK 1
fbInverter(
    bEnable := bEnable,
    bEStop := bEStop,
    bRun := bSorterEngine,
    bJogBackward := TRUE,
    sStationName := sStationName,
    udiSetVelocity := 600,
    udiActualVelocity := InEngineVelocityCV,
    uiStatusWord := InEngineSTW,
    uiControlWord => QnEngineCTW,
    udiTargetVelocity => QnEngineVelocitySV); // FB_MitsubishiInverter
END_ACTION

ACTION ACT_ManualMovements:
//W trybie ruchów manualnych wykonuj ruchy za pomocą rozkazów manualnych

rtbSeparator1				(CLK:=bManualSeparator1				, Q=>);	IF rtbSeparator1.Q				THEN bManualSeparator2				;END_IF	         	
rtbSeparator2				(CLK:=bManualSeparator2				, Q=>);	IF rtbSeparator2.Q				THEN bManualSeparator1			    ;END_IF     
rtbSleve1SeparatorActIn	    (CLK:=bManualSleve1SeparatorActIn	, Q=>);	IF rtbSleve1SeparatorActIn.Q	THEN bManualSleve1SeparatorActOut	;END_IF  
rtbSleve1SeparatorActOut    (CLK:=bManualSleve1SeparatorActOut	, Q=>);	IF rtbSleve1SeparatorActOut.Q 	THEN bManualSleve1SeparatorActIn    ;END_IF
rtbSleve2SeparatorActIn	    (CLK:=bManualSleve2SeparatorActIn	, Q=>);	IF rtbSleve2SeparatorActIn.Q	THEN bManualSleve2SeparatorActOut	;END_IF 
rtbSleve2SeparatorActOut    (CLK:=bManualSleve2SeparatorActOut	, Q=>);	IF rtbSleve2SeparatorActOut.Q 	THEN bManualSleve2SeparatorActIn    ;END_IF



IF NOT bRun THEN
	
	bHeightMotorUp				:= bManualHeightMotorUp;
	bHeightMotorDown			:= bManualHeightMotorDown;
	bSorterEngine				:= bManualSorterEngine;
	bBlow1						:= bManualSorterAir;
	bSleeveBlow					:= bManualSorterAir;
	bStopper1					:= bManualStopper;
	bStopper2					:= bManualStopper2;	
    bSeparator1					:= bManualSeparator1;			
    bSeparator2					:= bManualSeparator2;
    bSleve1SeparatorActIn		:= bManualSleve1SeparatorActIn;    
    bSleve1SeparatorActOut	    := bManualSleve1SeparatorActOut;
    bSleve2SeparatorActIn	    := bManualSleve2SeparatorActIn;
    bSleve2SeparatorActOut	    := bManualSleve2SeparatorActOut;
    bHammer1				    := bManualHammer1;          
    bHammer2				    := bManualHammer2;  
	bFormPositioning			:= bManualFormPositioning;        

END_IF


IF bHoming OR bHeightSet THEN
	eState:=E_Station.eHoming;
END_IF

IF bRun THEN	
	ACT_Running();
END_IF

//Zabezpieczenie przed kolizją stacji poprzez ruch podnośnika	
IF bHeightMotorDown AND lrHeightMotorCV<=lrMinHeight AND NOT bHoming AND NOT bHeightSet THEN
	bHeightMotorDown:=FALSE;
END_IF	

IF bHeightMotorUp AND lrHeightMotorCV>=lrMaxHeight AND NOT bHoming AND NOT bHeightSet THEN
	bHeightMotorUp:=FALSE;
END_IF
END_ACTION

ACTION ACT_ResetCommands:
//Reset komend ruchu 	


			bSorterEngine				:=	FALSE;
			bHeightMotorUp				:=	FALSE;
			bHeightMotorDown			:=	FALSE;
			bStopper1					:= FALSE;
			bStopper2					:= TRUE;			
 			//bSeparator1					:= FALSE;
 			//bSeparator2					:= FALSE;
 			//bSleve1SeparatorActIn		:= FALSE;  
 			//bSleve1SeparatorActOut	    := FALSE;
 			//bSleve2SeparatorActIn	    := FALSE;
 			//bSleve2SeparatorActOut	    := FALSE;
 			bHammer1				    := FALSE;
 			bHammer2				    := FALSE;
			bBlow1						:= FALSE;
			bSleeveBlow					:= FALSE;
			bFormPositioning			:= FALSE;
END_ACTION

ACTION ACT_Running:
//Obsługa sortera knotów - podawanie do separatora
CASE eRunningStateFeeder OF
	
	//NIEGOTOWY
	E_WickFeederSorterState.eDisabled:
		eRunningStateFeeder:=E_WickFeederSorterState.eReady;

	E_WickFeederSorterState.eReady:
		iTryUnblockWheel		:=	0;
		bTryUnblockWheel		:= FALSE;	
		fbInverter.bDirection 	:= TRUE;
		IF bRun THEN
			eRunningStateFeeder			:=E_WickFeederSorterState.eSorting;
		END_IF
	
	E_WickFeederSorterState.eSorting:
		bSorterEngine:=tonAirBeforeStart.Q;
		bBlow1:=TRUE;
		(*Próba odblokowania koła*)
			iTryUnblockWheel := iTryUnblockWheel + 1;
			IF rtWheelSensor.Q THEN
				iTryUnblockWheel	:=	0;
			END_IF
			IF tonEngineBlocked.Q THEN
				bTryUnblockWheel := TRUE;
			END_IF	
			IF bTryUnblockWheel THEN
				fbInverter.bDirection := FALSE;
			END_IF
			IF tonTryUnblockWheel.Q THEN
				iTryUnblockWheel		:=	0;//dp
				bTryUnblockWheel		:= FALSE;
				fbInverter.bDirection 	:= TRUE;
			END_IF

		(* Koniec Podawanie do toru jeden lub dwa*)		
						
		IF tonSortingEngineOff.Q THEN 
			eRunningStateFeeder 			:=E_WickFeederSorterState.eSleeveFull;
		END_IF
	
	E_WickFeederSorterState.eSleeveFull:
		bSorterEngine:=FALSE;
 		bBlow1:=NOT tonAirAfterStop.Q;
		IF tonAirAfterStop.Q THEN
			IF tonSortingEngineOn.Q THEN
				eRunningStateFeeder		:=E_WickFeederSorterState.eSorting; 
			END_IF
		END_IF
	
	E_WickFeederSorterState.eSleeveLowLevel:
		bSorterEngine:=TRUE;
		bBlow1:=TRUE;
		IF tonSortingEngineOff.Q THEN
			eRunningStateFeeder		 	:=E_WickFeederSorterState.eSorting;
		END_IF
	
END_CASE


		(* Koniec Próba odblokowania koła*)		
		CASE iSortingCase OF
			0:
				iSortingCase := iSortingCase	+	10;
				
			10:
				bStopper1:= TRUE;
				bStopper2:= TRUE;
				
				IF	bQueFullSensor THEN
					iSortingCase := iSortingCase	+	10;
				END_IF
				
			20:	
				bStopper1	:= FALSE;
				bStopper2	:= TRUE;
				IF tonCaseA.Q  AND NOT bWickBlocked THEN
					IF NOT fbbQueFullAtSleve1.bOUT AND (NOT bSeparatorLast OR fbbQueFullAtSleve2.bOUT) THEN
							bSeparator1			:= FALSE;
							bSeparator2			:= TRUE;
							IF tonbSeparatorPos2.Q THEN
								iSortingCase := iSortingCase	+	10;
								bSeparatorLast		:= TRUE;
							END_IF
					ELSIF NOT fbbQueFullAtSleve2.bOUT THEN	
							bSeparator1			:= TRUE;
							bSeparator2			:= FALSE;	
							IF tonbSeparatorPos1.Q THEN
								iSortingCase := iSortingCase	+	10;
								bSeparatorLast	:= FALSE;
							END_IF
					END_IF
				ELSIF tonCaseA.Q THEN
					iSortingCase := iSortingCase	+	10;
					bWickBlocked := FALSE;
				END_IF
									
			30:
				iSortingCase := iSortingCase	+	5;

			35:
				bSleeveBlow := TRUE;
				bStopper1	:= TRUE;
				bStopper2	:= FALSE;
				IF tonCaseB.Q AND fbbWickAtPipe.bOUT THEN
					bSleeveBlow  := FALSE;
					iSortingCase := iSortingCase	+	5;
				ELSIF fbbNotWickAtPipe.bOUT THEN
					bSleeveBlow  := FALSE;
					bWickBlocked := TRUE;
					iSortingCase := 10;
				END_IF	
				
			40:
				IF bSeparatorPos1 THEN
						bSeparator1			:= FALSE;
						bSeparator2			:= TRUE;
						iSortingCase		 := iSortingCase	+	10;
				ELSIF bSeparatorPos2 THEN
						bSeparator1			:= TRUE;
						bSeparator2			:= FALSE;		
						iSortingCase	 	:= iSortingCase	+	10;				
				END_IF

			50:	
				IF bSeparator2 AND tonbSeparatorPos2.Q THEN
					iSortingCase	 	:= 0;
				ELSIF bSeparator1 AND tonbSeparatorPos1.Q THEN
					iSortingCase	 	:= 0;				
				END_IF

		END_CASE
		(* Podawanie do toru jeden lub dwa*)


//Obsługa wbijaka 1
CASE eRunningState1 OF
	E_WickFeederState.eDisabled:
		eRunningState1					:= E_WickFeederState.eReady;
	E_WickFeederState.eFilling:
		;
	E_WickFeederState.eReady:	
		IF bWickAtSleve1 AND bRun1 AND NOT bCycleDone1 THEN
			eRunningState1				:= E_WickFeederState.ePuttingWick;
		END_IF
		IF NOT bRun1 THEN
			bCycleDone1 				:= FALSE;
			bCycleNotDone1 				:= FALSE;	
		END_IF
	E_WickFeederState.ePuttingWick:
		bSleve1SeparatorActIn			:= FALSE;			
		bSleve1SeparatorActOut			:= TRUE;
		IF bSleve1SeparatorOut THEN
			bHammer1					:= TRUE;
		END_IF
		//Jak siłownik dojdzie do końca ruchu - DODAĆ czasówkę
		IF tonHammer1Down.Q THEN
			bHammer1					:= FALSE;
			eRunningState1				:= E_WickFeederState.eWickPutted;
		END_IF
		IF NOT bRun1 THEN
			eRunningState1				:= E_WickFeederState.eReady;
		END_IF	
	E_WickFeederState.eWickPutted:
		bCycleDone1:=TRUE;
		IF bHammer1Up THEN
			bSleve1SeparatorActIn		:= TRUE;			
			bSleve1SeparatorActOut		:= FALSE;
			IF tobbSleve1SeparatorIn.Q THEN
				eRunningState1			:= E_WickFeederState.eReady;
			END_IF	
		END_IF
END_CASE	


//Obsługa wbijaka 2
CASE eRunningState2 OF
	E_WickFeederState.eDisabled:
		eRunningState2					:= E_WickFeederState.eReady;
		
	E_WickFeederState.eFilling:
		;
		
	E_WickFeederState.eReady:
		IF bWickAtSleve2 AND bRun2 AND NOT bCycleDone2 THEN
			eRunningState2			:= E_WickFeederState.ePuttingWick;
		END_IF
		IF NOT bRun2 THEN
			bCycleDone2 				:= FALSE;
			bCycleNotDone2 				:= FALSE;	
		END_IF	
		
	E_WickFeederState.ePuttingWick:
		bSleve2SeparatorActIn			:= FALSE;			
		bSleve2SeparatorActOut			:= TRUE;
		IF bSleve2SeparatorOut THEN
			bHammer2					:= TRUE;
		END_IF

		//Jak siłownik dojdzie do końca ruchu - DODAĆ czasówkę
		IF tonHammer2Down.Q  THEN
			bHammer2					:= FALSE;
			eRunningState2				:= E_WickFeederState.eWickPutted;
		END_IF
		IF NOT bRun2 THEN
			eRunningState2				:= E_WickFeederState.eReady;
		END_IF
		
	E_WickFeederState.eWickPutted:
		bCycleDone2:=TRUE;
		IF bHammer2Up THEN
			bSleve2SeparatorActIn		:= TRUE;			
			bSleve2SeparatorActOut		:= FALSE;
			IF tobbSleve2SeparatorIn.Q THEN
				eRunningState2			:= E_WickFeederState.eReady;
			END_IF	
		END_IF
END_CASE
END_ACTION

ACTION ACT_RunningHammer:
		IF bWickAtSleve1 AND bRun1 AND NOT bCycleDone1 THEN
			bSleve1SeparatorActIn		:= FALSE;			
			bSleve1SeparatorActOut		:= TRUE;
			IF bSleve1SeparatorOut THEN
				bHammer1				:= TRUE;
				eRunningState1			:= E_WickFeederState.ePuttingWick;
			END_IF
		END_IF

		IF NOT bRun1 THEN
			bCycleDone1 		:= FALSE;
			bCycleNotDone1 		:= FALSE;	
		END_IF
END_ACTION

ACTION ACT_Signals:
(** Timery na potrzeby bazowania**)
rtEncoderHomed(CLK:=bHeightMotorEncoderHomed,Q=>);
tonHeightNoChange(IN:=((bHeightMotorUp OR bHeightMotorDown OR tonHomingSensor.Q) AND (lrLastPositionHeightCV=lrHeightMotorCV)), PT:=T#2000MS); 
tonLimitPosMinReachedDelay(IN:=(lrHeightMotorCV<=lrMinHeight) AND eState=E_Station.eHoming,PT:=T#2S);
tonLimitPosMaxReachedDelay(IN:=(lrHeightMotorCV>=lrMaxHeight) AND eState=E_Station.eHoming,PT:=T#2S);
	
(** Timery używane podczas pracy stacji**)
tonSortingEngineOff(IN:=((eRunningStateFeeder=E_WickFeederSorterState.eSorting OR eRunningStateFeeder=E_WickFeederSorterState.eSleeveLowLevel) AND bRun AND bQueFullSensor),PT:=INT_TO_TIME(iTimeDelayOff));
tonSortingEngineOn(IN:=((eRunningStateFeeder=E_WickFeederSorterState.eSorting OR eRunningStateFeeder=E_WickFeederSorterState.eSleeveFull) AND bRun AND NOT bQueFullSensor),PT:=INT_TO_TIME(iTimeDelayOn));
tonSleeveFullEngineOn(IN:=(eRunningStateFeeder=E_WickFeederSorterState.eSleeveFull AND bRun AND NOT bQueFullSensor),PT:=INT_TO_TIME(iTimeDelayOff));
rtWheelSensor(CLK:=bWheelSensor, Q=>);
tonEngineBlocked(IN:=iTryUnblockWheel > 1500 AND bSorterEngine AND NOT bTryUnblockWheel,PT:=T#1MS); //Zablokowany silnik
tonTryUnblockWheel(IN:=bTryUnblockWheel, PT:=T#1S900MS);
//tofWickFeederSorterCapSensor(IN:=tonCapFeederSorterCapSensor.Q,PT:=T#100MS); //bylo 200
//tonCapFeederSorterCapSensor(IN:=bSorterCapSensor,PT:=T#3mS);//było 3ms
tonAirBeforeStart(IN:=eRunningStateFeeder=E_WickFeederSorterState.eSorting, PT:=T#1S);
//rtCapFeederSorterCapSensor(CLK:=tofCapFeederSorterCapSensor.Q,Q=>);

tonAirBeforeStart2(IN:=eRunningStateFeeder=E_WickFeederSorterState.eSorting, PT:=T#2S);
tonAirAfterStop(IN:=eRunningStateFeeder=E_WickFeederSorterState.eSleeveFull, PT:=T#2S);

tonbSeparatorPos1AndNotbWickAtSleve1(IN:=bSeparatorPos1 AND NOT bWickAtSleve1,PT:=T#3S);
tonbSeparatorPos2AndNotbWickAtSleve2(IN:=bSeparatorPos2 AND NOT bWickAtSleve2,PT:=T#3S);
tonbSeparatorPos1(IN:=bSeparatorPos1,PT:=T#300MS);
tonbSeparatorPos2(IN:=bSeparatorPos2,PT:=T#300MS);

tobbSleve1SeparatorIn(IN:=bSleve1SeparatorIn,PT:=T#1S);
tobbSleve2SeparatorIn(IN:=bSleve2SeparatorIn,PT:=T#1S);
fbbQueFullAtSleve1 (bIN:=	bQueFullAtSleve1,	tFilterTimeOn:=T#300MS, tFilterTimeOff:=T#300MS, 	bOUT=> );										
fbbQueFullAtSleve2 (bIN:=	bQueFullAtSleve2,	tFilterTimeOn:=T#300MS, tFilterTimeOff:=T#300MS, 	bOUT=> );										
fbbWickAtPipe 		(bIN:=	bWickAtPipe,		tFilterTimeOn:=T#100MS, tFilterTimeOff:=T#30MS,		bOUT=> );	
fbbNotWickAtPipe 	(bIN:=	NOT bWickAtPipe AND iSortingCase=35,		tFilterTimeOn:=T#2S, tFilterTimeOff:=T#100MS,		bOUT=> );	
									
tonCaseA			(IN:=iSortingCase = 20 , PT:=T#600MS);
tonCaseB			(IN:=iSortingCase = 35 , PT:=T#300MS);
tonCaseC			(IN:=iSortingCase = 20 , PT:=T#600MS);
tonCaseD			(IN:=iSortingCase = 20 , PT:=T#600MS);
//prszesunęcie wartosci czujnika po buforu opoznenia 

TimerOn (IN := NOT bImpOn, PT := T#10MS);
IF TimerOn.Q THEN
	bImpOn := TRUE;
END_IF
TimerOff (IN := bImpOn, PT := T#10MS);
IF TimerOff.Q THEN
	bImpON := FALSE;
END_IF

tonHammer1Down(IN:= bHammer1Down, PT:=T#200MS);
tonHammer2Down(IN:= bHammer2Down, PT:=T#200MS);

(** Dodatkowy timer przy zatrzymywaniu**)
tonStoppingTime( IN:= eState= E_Station.eStopping, PT:=T#2S);
END_ACTION

ACTION ACT_Warning:
 //Warning czujnik poziomu	
 	tonLowLevelSensor( IN:=( NOT  bWheelLevelSensor (*OR NOT bQueFullAfterWheelSensor*) OR NOT bQueFullSensor) AND bRun, PT:= T#5S);
 	
 	IF tonLowLevelSensor.Q THEN
 		bWarning				:= TRUE;
	ELSE
		bWarning				:= FALSE;
 	END_IF
END_ACTION

END_FUNCTION_BLOCK

(* stored: Version 1.2.0.0, ProductVersion 3.1.4026.13, FileIdentifier e7ee6229624cc21d0ee6a17dc6a17618cbd20523, FileSignature 13a131ac04f9de278d3e4888ad00071729109c0296af673369c2bef95be93959e503da5809fda02bc432a8ed99fe266445b20324541c74f72fac200b6a3c1f00be3946457e787848249a2f1f63ec669b506795072f0f47089f550b0b9bbcbd74c9e9b82e1237058e6a0d7bf1009c7a0e0e6e40d650b89ef499b0fc85ab7035861488e8691463a6a1725996c2d83b20f1328da542154d72246345aa6c26b7b66dd1eb4ecf56b1b8be35472eec8c7a771996412f48e37c212ef9726d9617eb61190fcc13b1ff8a707b45bf3efdcf1196a0e9dad65d7c10a01fe2d0671cd55b2fdfdf04b17ab6932181534d0723cad797561a546eebdb98ad8dc393671ab5ecd3a7
   POU FB_WickFeederStation: Id {eac517d9-c1aa-41cd-b728-14f6b5fca407}, SpecialFunc None
   Action ACT_Control: Id {19a029e0-b4d2-4e8e-bd52-aaad0a2064c2}
   Action ACT_ErrorHandling: Id {abe26291-ed0f-4a33-8ec3-c64a51933ba4}
   Action ACT_HeightMotor: Id {77521788-e1b8-4ad5-9e56-00a6cb09f2e0}
   Action ACT_Homing: Id {f91cb3d6-0030-45bc-baee-2ccec257ee0f}
   Action ACT_Inverter: Id {736cee0f-7518-4bbd-8c02-c171187a318e}
   Action ACT_ManualMovements: Id {6ec06beb-6726-41a3-8531-d2fa49d91982}
   Action ACT_ResetCommands: Id {8b39083c-2fac-459e-addf-f9ddc2eee9df}
   Action ACT_Running: Id {d9ad1dfe-142c-4860-b1d1-4860f582bc9d}
   Action ACT_RunningHammer: Id {7ce6b818-0f80-4ead-b3c8-965db961dd17}
   Action ACT_Signals: Id {4ac65e93-eb55-4872-aa6c-c3782d2b9b7b}
   Action ACT_Warning: Id {dce44a34-ee44-48c2-b41f-b80167e05ebf} *)
